// TwinCAT 3 PLC project cookie_module_shell
// ProgramVersion: 3.1.0.8
// libraries:
//   Tc2_Standard, * (Beckhoff Automation GmbH)
//   Tc2_System, * (Beckhoff Automation GmbH)
//   Tc3_Interfaces, * (Beckhoff Automation GmbH)
//   Tc3_Module, * (Beckhoff Automation GmbH)
//   Tc2_MC2,3.3.8.0,Beckhoff Automation GmbH
//   Tc2_TcpIp,3.3.2.0,Beckhoff Automation GmbH
//   Tc2_Utilities,3.3.7.0,Beckhoff Automation GmbH
// project tree:
//   DUTs/industrialPhysics/ MNG_APPLICATION_INPUTS_32BIT.TcDUT, MNG_APPLICATION_OUTPUTS_32BIT.TcDUT, MNG_DataArray.TcDUT (not stored), MNG_DatagramHeader.TcDUT (not stored), MNG_DatagramType.TcDUT (not stored), MNG_POSE6.TcDUT (not stored), MNG_RawDatagram.TcDUT (not stored), MNG_TRAFO.TcDUT (not stored), VEC3.TcDUT (not stored)
//   DUTs/InternalDataTypes/ eMainState.TcDUT, eSubState.TcDUT (not stored)
//   DUTs/OPC Interface/Server DUTs/ DUT_MODE.TcDUT, DUT_PARAMETER_INPUT.TcDUT, DUT_PARAMETER_OUTPUT.TcDUT, DUT_SERVER_MODULE_INTERFACE.TcDUT, DUT_SERVER_MODULE_INTERFACE_INPUT.TcDUT, DUT_SERVER_MODULE_INTERFACE_OUTPUT.TcDUT, DUT_SERVER_PARAMETERINPUTARRAY.TcDUT, DUT_SERVER_PARAMETEROUTPUTARRAY.TcDUT, DUT_SERVER_SKILLINPUTARRAY.TcDUT, DUT_SERVER_SKILLOUTPUTARRAY.TcDUT, DUT_SERVER_SKILL_INPUT.TcDUT, DUT_SERVER_SKILL_OUTPUT.TcDUT, DUT_SERVER_STATEVALUEARRAY.TcDUT, DUT_STATEVALUES.TcDUT
//   GVLs/ GVL.TcGVL, MI5.TcGVL, MNG_GLOBALS.TcGVL (not stored), OPCConstants.TcGVL
//   / PlcTask.TcTTO (not stored), SimuTask.TcTTO
//   POUs/ FB_EmergencyStop.TcPOU, FB_Error.TcPOU, FB_Init.TcPOU, FB_Output.TcPOU, FB_Ready.TcPOU, FB_Refill.TcPOU, FB_ResetSystem.TcPOU, FB_Separation.TcPOU, FB_Timer.TcPOU, FB_TurnDiskModulo.TcPOU, FB_TurnDiskToSensor.TcPOU, MAIN.TcPOU, FB_StorageLevel.TcPOU, FB_ResetAxis.TcPOU
//   POUs/industrialPhysics/ FB_LogFifo.TcPOU, MAIN_simu.TcPOU, MNG_SIMULATION.TcPOU, MNG_UPDATEIOS.TcPOU
// real-time tasks:
//   TASK PlcTask: cycle T#10ms, priority 20, ADS port 350
//   TASK SimuTask: cycle T#10ms, priority 21, ADS port 351
// motion (NC):
//   TASK NC-Task 1 SAF: cycle T#1ms, priority 4, ADS port 501
//   TASK NC-Task 1 SVB: cycle T#10ms, priority 8, ADS port 511
//   AXIS Axis 2 (id 2)
//     General: UnitName=Degree, UnitFlags=#x00000004
//     Dynamic: Acceleration=19710, Deceleration=19710, Jerk=59130
//     Velo: RefSearch=131.4, RefSync=131.4, SlowManual=657, FastManual=3942, Fast=13140, Maximum=13140
//     OtherSettings: AllowMotionCmdToSlave=true
//     encoder EncType=19
//       EncPara: ScaleFactorNumerator=360, ScaleFactorDenominator=1048576, MaxCount=#xffffffff
//         TimeComp: TimeCompMode=1
//     drive DrvType=16
//       DrvPara: MaxCount=#xffffffff
//         Analog: VeloReferenz=14454, VeloScale=32
//         TimeComp: TimeCompMode=1, TaskDelayCycles=1
//     controller CtrType=1
//       CtrPara: PriorControlFactor=1
//         PosDiffControl: Range=8, Time=0.3
//         PID: PosKp=25
//         Observer: BandWidth=20
// I/O:
//   DEVICE Device 1 (EtherCAT), AmsNetId 5.26.6.164.2.1
//     Term 1 (EK1200) [EK1200-5000 EtherCAT Power supply (2A E-Bus)]
//       Term 2 (EL1804) [EL1804 4Ch. Dig. Input 24V, 3ms]
//       Term 3 (EL2808) [EL2808 8Ch. Dig. Output 24V, 0.5A]
//       Term 4 (EL7211-0010) [EL7211-0010 1Ch. MDP742 Servo motor output stage with OCT (50V, 4.5A RMS)]
//       Term 5 (EK1110) [EK1110 EtherCAT extension]
//     Box 6 (ZAC50CN02 (Junction EtherCAT with PoE)) [ZAC50CN02 (Junction EtherCAT with PoE)]
//       Term 7 (Sub-Core 1 with two extern ports) [Sub-Core 1 with two extern ports]
//         Box 8 (OCPnnnP0150C) [OCPnnnP0150C Type 352]
//   DEVICE Device 3 (EtherCAT Automation Protocol) (disabled), AmsNetId 5.26.6.164.4.1
// variable links:
//   NC-Task 1 SAF/Axes/Axis 2 <-> Device 1 (EtherCAT)/Term 1 (EK1200)/Term 4 (EL7211-0010)
//     Enc/Inputs/In/nDataIn1 <-> FB Position/Position
//     Enc/Inputs/In/nDcInputTime <-> InfoData/DcInputShift
//     Drive/Inputs/In/nState1 <-> DRV Statusword/Statusword
//     Drive/Outputs/Out/nDataOut2 <-> DRV Target velocity/Target velocity
//     Drive/Inputs/In/nState2 <-> DRV Statusword/Statusword @bit 8
//     Drive/Inputs/In/nState4 @bit 1 <-> WcState/InputToggle
//     Enc/Inputs/In/nState4 @bit 1 <-> WcState/InputToggle
//     Drive/Inputs/In/nDcOutputTime <-> InfoData/DcOutputShift
//     Drive/Outputs/Out/nCtrl1 <-> DRV Controlword/Controlword
//     Enc/Inputs/In/nState4 <-> WcState/WcState
//     Drive/Outputs/Out/nCtrl2 <-> DRV Controlword/Controlword @bit 8
//     Drive/Inputs/In/nState4 <-> WcState/WcState
//   cookie_module_shell/cookie_module_shell Instance <-> Device 1 (EtherCAT)/Box 6 (ZAC50CN02 (Junction EtherCAT with PoE))
//     PlcTask Inputs/GVL.iDiskPosition <-> TxPDO/Read input 8 bit
//   cookie_module_shell/cookie_module_shell Instance <-> Device 1 (EtherCAT)/Box 6 (ZAC50CN02 (Junction EtherCAT with PoE))/Term 7 (Sub-Core 1 with two extern ports)/Box 8 (OCPnnnP0150C)
//     PlcTask Inputs/GVL.iStorageLevel <-> TxPDO/Measurement
//   cookie_module_shell/cookie_module_shell Instance <-> Device 1 (EtherCAT)/Term 1 (EK1200)/Term 2 (EL1804)
//     PlcTask Inputs/GVL.iCookieIntact <-> Channel 1/Input
//     PlcTask Inputs/GVL.iNoCookieInOutput <-> Channel 3/Input
//   cookie_module_shell/cookie_module_shell Instance <-> Device 1 (EtherCAT)/Term 1 (EK1200)/Term 3 (EL2808)
//     PlcTask Outputs/GVL.oTriggerCamera <-> Channel 1/Output
//   cookie_module_shell/cookie_module_shell Instance <-> NC-Task 1 SAF/Axes/Axis 2
//     PlcTask Inputs/GVL.axis.NcToPlc <-> Outputs/ToPlc
//     PlcTask Outputs/GVL.axis.PlcToNc <-> Inputs/FromPlc

CONFIGURATION cookie_module_shell
    RESOURCE PLC ON TwinCAT3
        TASK SimuTask(INTERVAL := T#10ms, PRIORITY := 21);
        PROGRAM MAIN_simu WITH SimuTask : MAIN_simu;
    END_RESOURCE
END_CONFIGURATION

// ---- DUTs/industrialPhysics/MNG_APPLICATION_INPUTS_32BIT.TcDUT

TYPE MNG_APPLICATION_INPUTS_32BIT :
STRUCT
    NumSignals                     : INT     := 5         ;
    HallSensor1_00_IR : BOOL    := 0; (* ysics/Keksmodul/Keksmodul - relevant/HallSensor1?IR *)
    HallSensor2_00_IR : BOOL    := 0; (* ysics/Keksmodul/Keksmodul - relevant/HallSensor2?IR *)
    init_sensor_cookie_module_00_IR : BOOL    := 0; (* l/Keksmodul - relevant/init_sensor_cookie_module?IR *)
    kein_cookie_mehr_00_IR : BOOL    := 0; (* /Keksmodul/Keksmodul - relevant/kein_cookie_mehr?IR *)
    cookiebox_sensor_00_IR : BOOL    := 0; (* Physics://physics/Keksmodul/cookiebox_sensor?IR *)
END_STRUCT
END_TYPE

// ---- DUTs/InternalDataTypes/eMainState.TcDUT
TYPE eMainState :
(
	init		:= 0,
	ready		:= 10,
	output		:= 20,
	separation	:= 30,
	refill		:= 40,
	emergencyStop	:= 50,
	error			:= 60,
	resetSystem		:= 70
);
END_TYPE

// ---- DUTs/industrialPhysics/MNG_APPLICATION_OUTPUTS_32BIT.TcDUT

TYPE MNG_APPLICATION_OUTPUTS_32BIT :
STRUCT
    NumSignals                     : INT     := 4         ;
    Disc_00_ACT_POS : REAL    := 0.0; (* ysics/Keksmodul/Keksmodul - relevant/Disc?KinActual *)
    A2014_09_12_Left_Predeterminado_00_ACT_POS : REAL    := 0.0; (* nt/Scissor/2014_09_12_Left_Predeterminado?KinActual *)
    A2014_09_12_Right_Predeterminado_00_ACT_POS : REAL    := 0.0; (* t/Scissor/2014_09_12_Right_Predeterminado?KinActual *)
    Keksquelle_00_TRIG02 : BOOL    := 0; (* Physics://physics/Keksmodul/Keksquelle?Trigger *)
END_STRUCT
END_TYPE

// ---- DUTs/OPC Interface/Server DUTs/DUT_MODE.TcDUT
/// MODE to run (inside of MODULE_INTERFACE_INPUT)
TYPE DUT_MODE :
(
	///Initialitzation number mode
	Init := 0,
	///Automatic number mode
	Auto := 1,
	///Manual number mode
	Manual := 2,
	Reset := 3
);
END_TYPE

// ---- DUTs/OPC Interface/Server DUTs/DUT_PARAMETER_INPUT.TcDUT
TYPE DUT_PARAMETER_INPUT :
STRUCT
	///Value of the parameter 
	Value: LREAL;
	///Possibility to a string value depending on the parameter
	StringValue: STRING(80);
END_STRUCT
END_TYPE

// ---- DUTs/OPC Interface/Server DUTs/DUT_PARAMETER_OUTPUT.TcDUT
TYPE DUT_PARAMETER_OUTPUT :
STRUCT
	///Free to use = TRUE, busy to use =FALSE
	Dummy: BOOL := TRUE;
	///ID of the parameter
	ID: UINT;
	///Name of the parameter
	Name: STRING(80);
	///Unit of the parameter
	Unit: STRING(80);
	///Optional parameter
	Required: BOOL;
	///Default parameter to work
	Default: LREAL;
	///Minimum value of the parameter
	MinValue: LREAL;
	///Maximum value of the parameter
	MaxValue: LREAL;
END_STRUCT
END_TYPE

// ---- DUTs/OPC Interface/Server DUTs/DUT_SERVER_MODULE_INTERFACE.TcDUT
/// MODULE INTERFACE INPUT AND OUTPUT 
TYPE DUT_SERVER_MODULE_INTERFACE :
STRUCT
	///Information that the module reads
	Input: DUT_SERVER_MODULE_INTERFACE_INPUT;
	///Information that the module write
	Output: DUT_SERVER_MODULE_INTERFACE_OUTPUT;
END_STRUCT
END_TYPE

// ---- DUTs/OPC Interface/Server DUTs/DUT_SERVER_MODULE_INTERFACE_INPUT.TcDUT
TYPE DUT_SERVER_MODULE_INTERFACE_INPUT :
STRUCT
	///Mode to run (init,auto,manual,..)
	Mode: INT;
	///check if the modules is alive
	ConnectionTestInput: BOOL;
	///Modules get their position
	PositionInput : LREAL;
	///Update data= TRUE, No updatedata=FALSE
	Watchbit: BOOL;
	///Emergency stop
	EmergencyStop: BOOL;
	///Range of INPUT skills
	SkillInput: DUT_SERVER_SKILLINPUTARRAY;
END_STRUCT
END_TYPE

// ---- DUTs/OPC Interface/Server DUTs/DUT_SERVER_MODULE_INTERFACE_OUTPUT.TcDUT
TYPE DUT_SERVER_MODULE_INTERFACE_OUTPUT :
STRUCT
	///Free to use = TRUE, busy to use =FALSE
	Dummy: BOOL := TRUE;
	///Individual name of the module
	Name: STRING(80);
	///Identification number of module
	ID: UINT;
	///IP address
	IP: STRING(80);
	///Show if the module is in Standby or not
	Idle: BOOL;
	///Show if the module is connected
	Connected: BOOL;
	///Feedback with conection test input
	ConnectionTestOutput: BOOL;
	///Show if the system has error when=TRUE
	Error: BOOL;
	///Identification number of the error
	ErrorID: UINT;
	///Description of the error
	ErrorDescription: STRING(80);
	///Description of the current task
	CurrentTaskDescription: STRING(80);
	///Position of the output
	PositionOutput: LREAL;
	/// Bool value of the Sensor
	PositionSensor: BOOL;
	///Range of OUTPUT skills
	SkillOutput: DUT_SERVER_SKILLOUTPUTARRAY;
	///Range of state values
	StateValue: DUT_SERVER_STATEVALUEARRAY;
END_STRUCT
END_TYPE

// ---- DUTs/OPC Interface/Server DUTs/DUT_SERVER_PARAMETERINPUTARRAY.TcDUT
TYPE DUT_SERVER_PARAMETERINPUTARRAY :
STRUCT
	ParameterInput0: DUT_PARAMETER_INPUT;
	ParameterInput1: DUT_PARAMETER_INPUT;
	ParameterInput2: DUT_PARAMETER_INPUT;
	ParameterInput3: DUT_PARAMETER_INPUT;
	ParameterInput4: DUT_PARAMETER_INPUT;
	ParameterInput5: DUT_PARAMETER_INPUT;
END_STRUCT
END_TYPE

// ---- DUTs/OPC Interface/Server DUTs/DUT_SERVER_PARAMETEROUTPUTARRAY.TcDUT
TYPE DUT_SERVER_PARAMETEROUTPUTARRAY :
STRUCT
	ParameterOutput0: DUT_PARAMETER_OUTPUT;
	ParameterOutput1: DUT_PARAMETER_OUTPUT;
	ParameterOutput2: DUT_PARAMETER_OUTPUT;
	ParameterOutput3: DUT_PARAMETER_OUTPUT;
	ParameterOutput4: DUT_PARAMETER_OUTPUT;
	ParameterOutput5: DUT_PARAMETER_OUTPUT;
END_STRUCT
END_TYPE

// ---- DUTs/OPC Interface/Server DUTs/DUT_SERVER_SKILLINPUTARRAY.TcDUT
TYPE DUT_SERVER_SKILLINPUTARRAY :
STRUCT
	SkillInput0: DUT_SERVER_SKILL_INPUT;
	SkillInput1: DUT_SERVER_SKILL_INPUT;
	SkillInput2: DUT_SERVER_SKILL_INPUT;
	SkillInput3: DUT_SERVER_SKILL_INPUT;
	SkillInput4: DUT_SERVER_SKILL_INPUT;
	SkillInput5: DUT_SERVER_SKILL_INPUT;
	SkillInput6: DUT_SERVER_SKILL_INPUT;
	SkillInput7: DUT_SERVER_SKILL_INPUT;
	SkillInput8: DUT_SERVER_SKILL_INPUT;
	SkillInput9: DUT_SERVER_SKILL_INPUT;
	SkillInput10: DUT_SERVER_SKILL_INPUT;
	SkillInput11: DUT_SERVER_SKILL_INPUT;
	SkillInput12: DUT_SERVER_SKILL_INPUT;
	SkillInput13: DUT_SERVER_SKILL_INPUT;
	SkillInput14: DUT_SERVER_SKILL_INPUT;
	SkillInput15: DUT_SERVER_SKILL_INPUT;
END_STRUCT
END_TYPE

// ---- DUTs/OPC Interface/Server DUTs/DUT_SERVER_SKILLOUTPUTARRAY.TcDUT
TYPE DUT_SERVER_SKILLOUTPUTARRAY :
STRUCT
	SkillOutput0: DUT_SERVER_SKILL_OUTPUT;
	SkillOutput1: DUT_SERVER_SKILL_OUTPUT;
	SkillOutput2: DUT_SERVER_SKILL_OUTPUT;
	SkillOutput3: DUT_SERVER_SKILL_OUTPUT;
	SkillOutput4: DUT_SERVER_SKILL_OUTPUT;
	SkillOutput5: DUT_SERVER_SKILL_OUTPUT;
	SkillOutput6: DUT_SERVER_SKILL_OUTPUT;
	SkillOutput7: DUT_SERVER_SKILL_OUTPUT;
	SkillOutput8: DUT_SERVER_SKILL_OUTPUT;
	SkillOutput9: DUT_SERVER_SKILL_OUTPUT;
	SkillOutput10: DUT_SERVER_SKILL_OUTPUT;
	SkillOutput11: DUT_SERVER_SKILL_OUTPUT;
	SkillOutput12: DUT_SERVER_SKILL_OUTPUT;
	SkillOutput13: DUT_SERVER_SKILL_OUTPUT;
	SkillOutput14: DUT_SERVER_SKILL_OUTPUT;
	SkillOutput15: DUT_SERVER_SKILL_OUTPUT;
END_STRUCT
END_TYPE

// ---- DUTs/OPC Interface/Server DUTs/DUT_SERVER_SKILL_INPUT.TcDUT
TYPE DUT_SERVER_SKILL_INPUT :
STRUCT
	///Range of parameters
	ParameterInput: DUT_SERVER_PARAMETERINPUTARRAY;
	///Start process
	Execute: BOOL;
END_STRUCT
END_TYPE

// ---- DUTs/OPC Interface/Server DUTs/DUT_SERVER_SKILL_OUTPUT.TcDUT
TYPE DUT_SERVER_SKILL_OUTPUT :
STRUCT
	///Free to use = TRUE, busy to use =FALSE
	Dummy: BOOL := TRUE;
	///Identification number of skill
	ID: UINT;
	///indentfication name of skill
	Name: STRING(80);
	///Skill activated
	Activated: BOOL;
	///Ready to do skill
	Ready: BOOL;
	///Skill in process
	Busy: BOOL;
	///Skill finish
	Done: BOOL;
	///Error in system
	Error: BOOL;
	///Range of parameters
	ParameterOutput: DUT_SERVER_PARAMETEROUTPUTARRAY;
END_STRUCT
END_TYPE

// ---- DUTs/OPC Interface/Server DUTs/DUT_SERVER_STATEVALUEARRAY.TcDUT
TYPE DUT_SERVER_STATEVALUEARRAY :
STRUCT
	StateValue0: DUT_STATEVALUES;
	StateValue1: DUT_STATEVALUES;
	StateValue2: DUT_STATEVALUES;
	StateValue3: DUT_STATEVALUES;
	StateValue4: DUT_STATEVALUES;
	StateValue5: DUT_STATEVALUES;
	StateValue6: DUT_STATEVALUES;
	StateValue7: DUT_STATEVALUES;
	StateValue8: DUT_STATEVALUES;
	StateValue9: DUT_STATEVALUES;
	StateValue10: DUT_STATEVALUES;
END_STRUCT
END_TYPE

// ---- DUTs/OPC Interface/Server DUTs/DUT_STATEVALUES.TcDUT
TYPE DUT_STATEVALUES :
STRUCT
	///Free to use = TRUE, busy to use =FALSE
	Dummy: BOOL := TRUE;
	///Value of the State
	Value: LREAL;
	///Name of the state
	Name: STRING(80);
	///Description of the state
	Description: STRING(80);
	///Unit of the state ()
	Unit: STRING(80);
END_STRUCT
END_TYPE

// ---- GVLs/GVL.TcGVL
VAR_GLOBAL
	pi : REAL := 3.14159;
																
	//<<Input Variables>>//
	//iExecute				AT%I*	: BOOL; 			// is there a order to separate cookies? --> from database
	//iClearence			AT%I*	: BOOL;				// did the user clear the refilling/maintenance process --> from HMI
														//@TODO: change to Mode change? mode: init, auto, manual
	//iEmergencyStop		AT%I*	: BOOL;				// stop all running tasks and transform the machine in a safe state
	
	iDiskPosition 		AT%I*	: INT; 				// is the gap of the disk at the storage? --> 2 the ramp? --> 1 --> from hall sensor
	iNoCookieInOutput	AT%I*	: BOOL;				// is the cookie in the ouput (on the clamp)? --> from light barrier sensor
	iStorageLevel 		AT%I*	: DINT;			// number of remaining cookies in the storage --> from distance sensor
	iCookieIntact		AT%I*	: BOOL;				// camera detection if cookie intact or broken
	

	//<<Output Variables>>//
	oTriggerCamera		AT%Q*	: BOOL	:= FALSE;	//Variable to init the flashing mode of the cam		
	
	//<<Internal Variables>>//
	mainState 					: eMainState		:= eMainState.init;
	refillSubState				: eSubState			:= eSubState.step0;
	separationSubState			: eSubState			:= eSubstate.step0;
	initSubState				: eSubState			:= eSubstate.step0;
	outputSubState				: eSubState			:= eSubstate.step0;
	emergencySubState			: eSubState			:= eSubstate.step0;
	errorSubState				: eSubState			:= eSubstate.step0;
	resetSubState				: eSubState			:= eSubstate.step0;

	axis	 					: AXIS_REF;
	empty						: BOOL;				// is cookie storage empty
	fastVel						: INT	:= 40;		//@TODO: Use something to change velocity in ParameterInput
	slowVel						: INT	:= 15;		//@TODO: Use something to change velocity in ParameterInput
	
	modulePositionInitialized	: BOOL := FALSE;	// is the module position initialized
	firstRun					: BOOL := TRUE;		// is this the first init? then wait for axis to get ready
	
	
	//<<For Simulation>>//
	offset						: LREAL;
	infinitsimu					: BOOL;
	infinitsimu2				: BOOL;
	init_sensor 				: BOOL;      //AT	%I*, muss vor :BOOL ,Änderung km
	SensorPosition				: LREAL;				
	
END_VAR

// ---- GVLs/MI5.TcGVL
VAR_GLOBAL
	//<<OPC-UA Module Interface>>//
	{attribute 'OPC.UA.DA' := '1'}
	Module2101 : DUT_SERVER_MODULE_INTERFACE;
	{attribute 'OPC.UA.DA' := '1'}
	reset : BOOL := FALSE;
	{attribute 'OPC.UA.DA' := '1'}
	cameraFix : BOOL := FALSE;
END_VAR

// ---- GVLs/OPCConstants.TcGVL
VAR_GLOBAL CONSTANT
	///Maximum number of skillparameters
	ParameterCnt: INT := 5;
	///Maximum number of skills per Module
	SkillCnt: INT := 15;
	///Maximum number of Statevalues of one Module
	StateCnt: INT := 10;
	///Maximum number of modules
	ModuleCnt: INT := 10;
	///Maximum number of Tasks in Production List
	TaskCnt: INT := 30;
	///Maximum number  of offered recipes
	OfferCnt: INT := 5;
	///Maximum number of Orders in Queue
	OrderCnt: INT := 5;
	///Number of user set parameters per recipe
	UserParameterCnt: INT := 5;
	///Number of skills per task
	TaskSkillCnt: INT := 50;
END_VAR

// ---- POUs/industrialPhysics/MAIN_simu.TcPOU

PROGRAM MAIN_simu
VAR
    simIO : MNG_Simulation;
END_VAR

// Update IOs with simulation
simIO(bEnable := TRUE);

// Application code follows here:

END_PROGRAM

// ---- POUs/industrialPhysics/MNG_SIMULATION.TcPOU
FUNCTION_BLOCK MNG_Simulation
VAR_INPUT
    bEnable    : BOOL                          := FALSE;
    outputs AT %I*   : MNG_Application_Outputs_32Bit         ;
END_VAR
VAR_OUTPUT
    inputs AT %Q*  : MNG_Application_Inputs_32Bit          ;
END_VAR
VAR
    ioUpdater  : MNG_UpdateIOs                 := (sRemoteHost := '192.168.42.31', nRemotePort := 5110);
    fbCloseAll : FB_SocketCloseAll;
    bCloseAll  : BOOL := TRUE;
	trig		: BOOL;
END_VAR

(* @END_DECLARATION := '0'                                                    *)
IF bCloseAll THEN (*On PLC reset or program download close all old (opened) connections *)
    bCloseAll := FALSE;
    fbCloseAll( bExecute:= TRUE );
ELSE
    fbCloseAll( bExecute:= FALSE );
END_IF

IF NOT fbCloseAll.bBusy THEN

    (* ------------------------------------- trigger data exchange ----------------------------------------------------------------------------*)
    ioUpdater(Outputs := outputs, Inputs := inputs, bEnable := bEnable);

END_IF

// Application code follows here:

{*IF GVL.infinitsimu THEN
	outputs.Disc_00_ACT_POS := (REAL_TO_INT(GVL.SensorPosition -180 + GVL.axis.NcToPlc.ModuloActPos))MOD 360;
ELSE
	IF GVL.infinitsimu2 THEN
		outputs.Disc_00_ACT_POS := (REAL_TO_INT(GVL.SensorPosition + GVL.axis.NcToPlc.ModuloActPos))MOD 360;
	ELSE
		outputs.Disc_00_ACT_POS := GVL.axis.NcToPlc.ModuloActPos;
	END_IF	
END_IF*}

outputs.Disc_00_ACT_POS := GVL.axis.NcToPlc.ModuloSetPos;

//storageLevel.full := inputs.kein_cookie_mehr_00_IR;

outputs.A2014_09_12_Right_Predeterminado_00_ACT_POS := ABS(SIN(((GVL.axis.NcToPlc.ActPos*pi)/180)))*(-7);
outputs.A2014_09_12_Left_Predeterminado_00_ACT_POS := ABS(SIN(((GVL.axis.NcToPlc.ActPos*pi)/180)))*(7);

//GVL.iNoCookieInOutput := inputs.cookiebox_sensor_00_IR;
//GVL.iDiskAtStorage := inputs.HallSensor1_00_IR;
//GVL.iDiskAtRamp := inputs.HallSensor2_00_IR;

GVL.init_sensor := inputs.cookiebox_sensor_00_IR;

IF GVL.mainState = eMainState.ready THEN
	trig := TRUE;
ELSE 
	trig := FALSE;
END_IF

//trigger(CLK:= trig, Q=> newCookie);
IF trig THEN
	outputs.Keksquelle_00_TRIG02 := TRUE;
ELSE 
	outputs.Keksquelle_00_TRIG02 := FALSE;
END_IF 


//outputs.Keksquelle_00_ReleaseTime := 60;
//outputs.Keksquelle_00_AlwaysOn := TRUE;

END_FUNCTION_BLOCK

// ---- POUs/industrialPhysics/MNG_UPDATEIOS.TcPOU
FUNCTION_BLOCK MNG_UpdateIOs
(* This function block implements simple TCP/IP client protocol.              *)
(* The max. size of binary tx/rx data has to be <= PLCPRJ_BUFFER_SIZE         *)
VAR_IN_OUT
    Outputs : MNG_Application_Outputs_32Bit;    (* Tx user data *)
    Inputs      : MNG_Application_Inputs_32Bit                        ; (* Rx user data *)
END_VAR

VAR_INPUT
    bDbg        : BOOL                         := FALSE               ; (* TRUE => Enable debug output, FALSE => Disable debug output *)
    sRemoteHost : STRING(15)                   := '127.0.0.1'         ; (* IP address of remote server *)	
    nRemotePort : UDINT                        := 5000                ; (* Remote server port *)
    bEnable     : BOOL                         := FALSE               ; (* TRUE => Enable/connect, FALSE => Disable/disconnect *)
    tReconnect  : TIME                         := T#5s                ;
END_VAR

VAR_OUTPUT
    errors      : FB_LogFifo                                          ; (* Error message fifo *)
    eState      : E_SocketConnectionState      := eSOCKET_DISCONNECTED; (* TCP/IP connection state *)
END_VAR

VAR
    counter          : DWORD                        := 0                   ;
    fbConnect        : FB_ClientServerConnection    := (tReconnect := T#5s); (* Create/release TCP/IP connection *)
    fbSend           : FB_SocketSend                                       ; (* Send TCP/IP data *)
    fbReceive        : FB_SocketReceive                                    ; (* Receive TCP/IP data *)
    state            : BYTE                                                ; (* Global state *)
    tx_state         : BYTE                                                ; (* Tx state *)
    rx_state         : BYTE                                                ; (* Rx state *)

    toServer         : MNG_RawDatagram                                     ;
    fromServer       : MNG_RawDatagram                                     ;
    cbReceived       : UDINT                                               ; (* Count of received data bytes *)
    cbRx             : UDINT                                               ; (* Rx frame byte size *)

    bDisconnect      : BOOL                                                ; (* Disconnect flag, if set the socket will be closed *)
    pollTimer        : TON                                                 ; (* Rx data poll timer *)
    bAbort           : BOOL                                                ; (* Flag to abort frame parsing loop *)
    sID              : STRING(20)                   := ''                  ;
    clock            : FB_LocalSystemTime           := ( bEnable := TRUE ) ; (* OS clock *)
    _byteCount       : DWORD                                               ;
    _i               : DWORD                                               ;
    _ptr             : POINTER TO BYTE                                     ;
    _internalInputs  : MNG_Application_Inputs_32Bit                        ;
    DWordBuffer      : DWORD                                               ; (* convert DWORD data *)
    DIntBuffer       : DINT                                                ; (* convert DINT data *)
END_VAR


(* refresh clock time                                                         *)
clock();

(* state chart                                                                *)
CASE state OF
    0:(* Init state *)
        (*rx.A_Reset(bDbg := bDbg)  ; (* Reset RX fifo (optional) *)
        tx.A_Reset    (bDbg := bDbg); (* Reset TX fifo (optional) *)*)
        errors.Clear(); (* Reset error fifo (optional) *)

        pollTimer( IN := FALSE, PT := PLCPRJ_RECEIVER_POLLING_CYCLE_TIME );
        bDisconnect := FALSE;(* Reset disconnect flag *)
        cbReceived  := 0;(* Reset number of received data bytes *)
        tx_state    := 0;(* Reset tx state machine *)
        rx_state    := 0;(* Reset rx state machine *)
        state       := 1;(* Go to the next step *)

    1:(* Create TCP/IP connection *)
        fbConnect(sSrvNetID := '',
                  nMode := CONNECT_MODE_ENABLEDBG,(* Enable debug output *)
                  sRemoteHost := sRemoteHost,
                  nRemotePort := nRemotePort,
                  tReconnect  := tReconnect,
                  bEnable     := bEnable,
                  eState      => eState);
        IF NOT fbConnect.bBusy THEN

            (* Create identification string used by debug messages *)
            sID          := CONCAT(CONCAT('[', DWORD_TO_HEXSTR(fbConnect.hSocket.handle, 4, FALSE) ), ']');
            errors.sMessage := CONCAT('CLI.Err', sID);

            IF NOT fbConnect.bError THEN
                IF eState = eSOCKET_CONNECTED THEN(* we are connected *)
                    state := 2;
                END_IF
            ELSE(* connect error: log error *)
                errors.Error(nErrId := fbConnect.nErrId);
            END_IF
        END_IF

    2:(* Data exchange state *)
        bDisconnect := NOT bEnable OR bDisconnect; (* user/internal disconnect requested? *)
        IF bDisconnect AND (tx_state = 0) AND (rx_state = 0) THEN
            state := 3;(* disconnect *)
        ELSE
            (*--------------------------- Send tx data -------------------------------------------*)
            CASE tx_state OF
                0:
                    IF NOT bDisconnect THEN

                        (* forcefully send data each cycle *)

                        (* create the raw datagram *)
                        _byteCount                   := 20;
                        toServer.Header.ByteCount    := HOST_TO_BE32(in := _byteCount);
                        toServer.Header.DatagramType := HOST_TO_BE32(in := MNG_Raw32BitImage);
                        toServer.Header.Counter      := Counter;

                        toServer.Payload[1] := HOST_TO_BE32(4); (* number of signals *)

                        (* FLOAT32 Disc_00_ACT_POS *)
                        MEMCPY(destAddr := ADR(DWordBuffer), srcAddr := ADR(Outputs.Disc_00_ACT_POS), n := 4);
                        toServer.Payload[2] := HOST_TO_BE32(DWordBuffer);

                        (* FLOAT32 A2014_09_12_Left_Predeterminado_00_ACT_POS *)
                        MEMCPY(destAddr := ADR(DWordBuffer), srcAddr := ADR(Outputs.A2014_09_12_Left_Predeterminado_00_ACT_POS), n := 4);
                        toServer.Payload[3] := HOST_TO_BE32(DWordBuffer);

                        (* FLOAT32 A2014_09_12_Right_Predeterminado_00_ACT_POS *)
                        MEMCPY(destAddr := ADR(DWordBuffer), srcAddr := ADR(Outputs.A2014_09_12_Right_Predeterminado_00_ACT_POS), n := 4);
                        toServer.Payload[4] := HOST_TO_BE32(DWordBuffer);

                        (* BOOL Keksquelle_00_TRIG02 *)
                        IF Outputs.Keksquelle_00_TRIG02 THEN
                            toServer.Payload[5] := 16#FFFFFFFF;   (*BOOL *)
                        ELSE
                            toServer.Payload[5] := 0;
                        END_IF;

                        toServer.Header.SentTime := HOST_TO_BE32(in := clock.systemTime.wMilliseconds + clock.systemTime.wMinute * 60000);

                        (* send frame *)
                        fbSend(bExecute  := FALSE);
                        fbSend(sSrvNetID := '',
                               hSocket   := fbConnect.hSocket,
                               cbLen     := SIZEOF(toServer.Header) + _byteCount,(* size of header + size of user data *)
                               pSrc      := ADR(toServer),(* pointer to the frame data *)
                               bExecute  := TRUE,
                               tTimeout  := T#5s);

                        tx_state := 1;
                    END_IF
                1:(* wait until send not busy *)
                    fbSend( bExecute := FALSE );
                    IF NOT fbSend.bBusy THEN
                        tx_state := 0;
                        IF NOT fbSend.bError THEN(* no error *)
                            ;
                        ELSE(* send error => log error and disconnect *)
                            errors.Error(nErrId := fbSend.nErrId );
                            bDisconnect := TRUE;(* set flag *)
                        END_IF
                    END_IF
            END_CASE

            (* ------------------------------------------- Get/fetch rx data ----------------------------------------------------------------- *)
            CASE rx_state OF
                0:
                    IF NOT bDisconnect THEN
                        pollTimer( IN := TRUE );
                        IF pollTimer.Q THEN
                            pollTimer( IN := FALSE );

                            fbReceive( bExecute := FALSE );
                            fbReceive( 	sSrvNetId	:= '',
                            hSocket		:= fbConnect.hSocket,
                            cbLen		:= SIZEOF(fromServer) - cbReceived,
                            pDest		:= ADR(fromServer) + cbReceived,
                            bExecute	:= TRUE,
                            tTimeout	:= T#5s );
                            rx_state := 1;
                        END_IF
                    END_IF
                1:(* wait until receive not busy *)
                    fbReceive( bExecute := FALSE );
                    IF NOT fbReceive.bBusy THEN
                        rx_state := 0;
                        IF NOT fbReceive.bError THEN
                            IF fbReceive.nRecBytes > 0 THEN (* some bytes received *)

                                pollTimer( PT := T#0s );(* increase polling speed *)
                                cbReceived := cbReceived + fbReceive.nRecBytes;

                                (* parse received bytes *)
                                REPEAT
                                    bAbort := TRUE;(* set flag *)
                                    IF cbReceived >= SIZEOF(fromServer.Header) THEN (* all header bytes received => check header data *)

                                        (* correct header data *)
                                        fromServer.Header.ByteCount    := BE32_TO_HOST(fromServer.Header.ByteCount);
                                        Counter                        := fromServer.Header.Counter;
                                        fromServer.Header.SentTime     := BE32_TO_HOST(fromServer.Header.SentTime);
                                        fromServer.Header.DatagramType := BE32_TO_HOST(fromServer.Header.DatagramType);

                                        IF (fromServer.Header.ByteCount <= SIZEOF( fromServer.Payload))(* check frame (user data) length *)
                                        THEN

                                            cbRx := SIZEOF(fromServer.Header) + fromServer.Header.ByteCount;(* calculate the (expected) length of the rx frame *)
                                            IF cbReceived >= cbRx  THEN (* all frame bytes received? *)

                                               (* currently only use the data on a 32 Bit raw image *)
                                                IF fromServer.Header.DatagramType = MNG_Raw32BitImage THEN

                                                    IF 20 = (fromServer.Header.ByteCount - 4) THEN

                                                        (* BOOL HallSensor1_00_IR *)
                                                        Inputs.HallSensor1_00_IR := fromServer.Payload[2]<>0;

                                                        (* BOOL HallSensor2_00_IR *)
                                                        Inputs.HallSensor2_00_IR := fromServer.Payload[3]<>0;

                                                        (* BOOL init_sensor_cookie_module_00_IR *)
                                                        Inputs.init_sensor_cookie_module_00_IR := fromServer.Payload[4]<>0;

                                                        (* BOOL kein_cookie_mehr_00_IR *)
                                                        Inputs.kein_cookie_mehr_00_IR := fromServer.Payload[5]<>0;

                                                        (* BOOL cookiebox_sensor_00_IR *)
                                                        Inputs.cookiebox_sensor_00_IR := fromServer.Payload[6]<>0;

                                                    ELSE(* receive error: invalid frame format/data *)
                                                        errors.Error(nErrId := PLCPRJ_ERROR_INVALID_IO_FORMAT_RECEIVED );
                                                    END_IF

                                                END_IF

                                                MEMMOVE( ADR( fromServer ), ADR( fromServer ) + cbRx,  cbReceived - cbRx );(* shift the remaining rx bytes *)
                                                cbReceived := cbReceived - cbRx;(* recalculate the size of the remaining rx bytes *)

                                                bAbort := FALSE;(* reset flag, try to parse next frame *)

                                                (* ELSE repeat reading *)
                                            END_IF

                                        ELSE(* receive error: invalid frame format/data *)
                                            errors.Error(nErrId := PLCPRJ_ERROR_INVALID_FRAME_FORMAT );
                                            bDisconnect := TRUE;(* set flag *)
                                        END_IF
                                        (* ELSE repeat reading *)
                                    END_IF (* IF cbReceived >= SIZEOF(rxFrame.head) THEN *)

                                UNTIL bAbort
                                END_REPEAT

                            ELSE(* fbReceive.nRecBytes = 0, repeat reading *)
                                pollTimer( PT := PLCPRJ_RECEIVER_POLLING_CYCLE_TIME );(* slow down the polling cycle *)
                            END_IF(* IF fbReceive.nRecBytes > 0 THEN *)
                        ELSE(* receive error => log error and disconnect *)
                            errors.Error(nErrId := fbReceive.nErrId );
                            bDisconnect := TRUE;(* set flag *)
                        END_IF

                    END_IF(*IF NOT fbReceive.bBusy THEN*)

            END_CASE

        END_IF

    3:(* disconnect *)
        fbConnect( bEnable:= FALSE, eState=>eState );
        IF eState = eSOCKET_DISCONNECTED THEN
            state := 0;
        END_IF

END_CASE

END_FUNCTION_BLOCK

// ---- POUs/industrialPhysics/FB_LogFifo.TcPOU
(* Log/debug/error message fifo *)
FUNCTION_BLOCK FB_LogFifo
VAR_INPUT
	bLog		: BOOL 		:= FALSE;(* TRUE => Enable log message output, FALSE => Disable *)
	sPrefix		: STRING 	:= 'Unknown::';(* Log message description string (allows the identification of log message source) *)
	
	sMessage	: STRING 	:= '';(* String message to add (write) to the fifo *)
	nErrID		: UDINT 	:= 0;(* Error code to add (write) to the fifo *)
	hSocket		: T_HSOCKET;(* Socket connection handle *)
END_VAR
VAR_OUTPUT
	bOk			: BOOL;(* TRUE = New entry added or removed succesfully, FALSE = Fifo overflow or fifo empty *)
	sGet		: T_MaxString := '';(* String entry removed (read) from fifo *)
	nCount		: UDINT := 0;(* Number of fifo entries *)
END_VAR
VAR
	fbBuffer 	: FB_StringRingBuffer;(* Basic (lower level) string buffer control function block *)
	buffer		: ARRAY[0..PLCPRJ_BUFFER_SIZE] OF BYTE;(* Internal buffer memory *)
	sSource		: T_MaxString;	
	sPut		: T_MaxString;
END_VAR

;

ACTION Error:
(* Adds new fifo entry *)
IF nErrID = 0 THEN
	sSource := '::Error: 0x';
ELSIF ( nErrID AND 16#80000000) = 16#80000000 THEN
	IF nErrID = 16#80072746 THEN
		sSource := '::Win32 error (the connection is reset by remote side): 0x';
	ELSE
		sSource := '::Win32 error: 0x';
	END_IF
ELSIF (nErrID AND 16#00008100) = 16#00008100 THEN
	CASE nErrID OF
		PLCPRJ_ERROR_RECEIVE_TIMEOUT:
			sSource := '::PLC sample project receive timeout error: 0x';
		PLCPRJ_ERROR_SENDFIFO_OVERFLOW:
			sSource := '::PLC sample project send fifo overflow error: 0x';
		PLCPRJ_ERROR_RECFIFO_OVERFLOW:
			sSource := '::PLC sample project receive fifo overflow error: 0x';
		PLCPRJ_ERROR_INVALID_FRAME_FORMAT:
			sSource := '::PLC sample project invalid frame format error: 0x';
	ELSE
		sSource := '::Other PLC sample project error: 0x';
	END_CASE
ELSIF (nErrID AND 16#00008000) = 16#00008000 THEN
	sSource := '::Internal TCP/IP Connection Server error: 0x';
ELSE
	sSource := '::TwinCAT System error: 0x';
END_IF

sPut := CONCAT( CONCAT( CONCAT( sPrefix, sMessage ), sSource ), DWORD_TO_HEXSTR( nErrID AND 16#FFFF, 0, FALSE ) ); 

fbBuffer.A_AddTail( pBuffer:= ADR(buffer), cbBuffer:= SIZEOF(buffer),
					putValue:= sPut, bOk=>bOk, nCount=>nCount );
IF bOk THEN
	IF bLog THEN(* Log error message *)
		ADSLOGSTR( ADSLOG_MSGTYPE_ERROR OR ADSLOG_MSGTYPE_LOG, '%s', sPut );	
	END_IF
END_IF
END_ACTION

ACTION Message:
(* Adds new fifo entry *)
sPut := CONCAT( CONCAT( sPrefix, sMessage ), CONCAT( '::', HSOCKET_TO_STRING(hSocket) ) );
fbBuffer.A_AddTail( pBuffer:= ADR(buffer), cbBuffer:= SIZEOF(buffer),
					putValue:= sPut, bOk=>bOk, nCount=>nCount );
IF bOk THEN
	IF bLog THEN(* Log information message *)
		ADSLOGSTR( ADSLOG_MSGTYPE_HINT OR ADSLOG_MSGTYPE_LOG, '%s', sPut );	
	END_IF
END_IF
END_ACTION

ACTION Remove:
(* Removes oldest fifo entry *)
IF nCount = 0 THEN
	sGet := '';
	bOk := FALSE;
	RETURN;
END_IF

fbBuffer.A_RemoveHead( pBuffer:= ADR(buffer), cbBuffer:= SIZEOF(buffer),
						getValue=>sGet, bOk=>bOk, nCount=>nCount );
END_ACTION

ACTION Clear:
(* Clears all fifo entries *)
fbBuffer.A_Reset( 	pBuffer := ADR( buffer ), cbBuffer := SIZEOF( buffer ), 
					bOk=>bOk, nCount=>nCount, getValue=>sGet );
END_ACTION

END_FUNCTION_BLOCK

// ---- POUs/FB_EmergencyStop.TcPOU
FUNCTION_BLOCK FB_EmergencyStop
VAR_INPUT
END_VAR
VAR_OUTPUT
END_VAR
VAR
END_VAR

CASE emergencySubState OF

	step0:	//setting of OPCUA variables
			Module2101.Output.SkillOutput.SkillOutput0.Busy := FALSE;
			Module2101.Output.SkillOutput.SkillOutput0.Done := FALSE;
			Module2101.Output.SkillOutput.SkillOutput0.Dummy := FALSE;
			Module2101.Output.SkillOutput.SkillOutput0.Error := TRUE;
			Module2101.Output.SkillOutput.SkillOutput0.Ready := FALSE;
			//go into the right error state
			Module2101.Output.ErrorID := 2;
			Module2101.Output.CurrentTaskDescription := 'Emergency stop';
			Module2101.Output.Error := TRUE;
			Module2101.Output.ErrorDescription := 'Emergency stop';
			
			//wait for process tool to set the module in manual mode
			IF(Module2101.Input.Mode = DUT_MODE.Manual) THEN
				emergencySubState := step1;
			END_IF
			
	step1:	//wait for process tool to set the module in init mode
			IF(Module2101.Input.Mode = DUT_MODE.Auto) THEN
				//reset error 
				Module2101.Output.Error := FALSE;
				Module2101.Output.ErrorDescription := '';
				Module2101.Output.ErrorID := 0;
				
				//change to init state
				initSubState := step0;
				mainState := eMainState.init;
				emergencySubState := step0;
			END_IF
			
			
	step2:	
			
	step3:	

END_CASE

END_FUNCTION_BLOCK

// ---- POUs/FB_Error.TcPOU
FUNCTION_BLOCK FB_Error
VAR_INPUT
END_VAR
VAR_OUTPUT
END_VAR
VAR
	resetAxis			: FB_ResetAxis;
END_VAR

//@TODO: implement all possible errors

CASE errorSubState OF

	step0:	Module2101.Output.SkillOutput.SkillOutput0.Busy := FALSE;
			Module2101.Output.SkillOutput.SkillOutput0.Done := FALSE;
			Module2101.Output.SkillOutput.SkillOutput0.Dummy := FALSE;
			Module2101.Output.SkillOutput.SkillOutput0.Error := TRUE;
			Module2101.Output.SkillOutput.SkillOutput0.Ready := FALSE;
			
			// Error: axis got stuck
			IF (axis.Status.ErrorID = 17744) THEN
				Module2101.Output.ErrorDescription := 'Axis got stuck. Please clear module.';
				Module2101.Output.ErrorID := 101;
				errorSubState := step1;
			END_IF
			
			IF (Module2101.Output.ErrorID = 0) THEN
				Module2101.Output.ErrorDescription := 'Unknown Error.';
				Module2101.Output.ErrorID := 199;
				errorSubState := step1;
			END_IF
			
			//change in the right error state
			Module2101.Output.CurrentTaskDescription := 'Error';
			Module2101.Output.Error := TRUE;
			
	step1:	//wait for process tool to set the module in manual mode
			IF(Module2101.Input.Mode = DUT_MODE.Manual) THEN
				resetAxis(execute:= FALSE);
				errorSubState := step2;
			END_IF
			
	step2:	IF NOT resetAxis.done THEN
				// axreset
				resetAxis (execute := TRUE);
			ELSE			
				errorSubState := step3;
			END_IF
			
	step3:	//wait for process tool to set the module in init mode
			IF(Module2101.Input.Mode = DUT_MODE.Auto) THEN
				
				//reset error 
				Module2101.Output.Error := FALSE;
				Module2101.Output.ErrorDescription := '';
				Module2101.Output.ErrorID := 0;
				
				//change to init state
				initSubState := step0;
				errorSubState := step0;
				mainState := eMainState.init;				
			END_IF
END_CASE

END_FUNCTION_BLOCK

// ---- POUs/FB_ResetAxis.TcPOU
FUNCTION_BLOCK FB_ResetAxis
VAR_INPUT
	execute: BOOL;
END_VAR
VAR_OUTPUT
	done : BOOL;
	busy : BOOL;
	error: BOOL;
END_VAR
VAR
	state			: INT := 0;
	fbreset			: Tc2_MC2.MC_Reset;
END_VAR

IF execute THEN
	CASE state OF
	
	0: 
		done := FALSE;
		fbreset(axis := axis, Execute := FALSE);
		state := 1;
		
	1:
		fbreset(
				Axis:= axis, 
				Execute:= TRUE, 
				Done=> , 
				Busy=> , 
				Error=> error, 
				ErrorID=> );
		IF fbreset.Done THEN
			state := 2;
		END_IF
		
	2:	
		execute := FALSE;
		done  := TRUE;
		state := 0;

	END_CASE
ELSE
	done := FALSE;
	state := 0;
END_IF

END_FUNCTION_BLOCK

// ---- POUs/FB_Init.TcPOU
FUNCTION_BLOCK FB_Init
VAR_INPUT
END_VAR
VAR_OUTPUT	
END_VAR
VAR
	turnDiskSensor	: FB_TurnDiskToSensor;		//turns disk to next sensor anti-clockwise
	turnDiskMod		: FB_TurnDiskModulo;		//turns disk back due to lag while stopping
	setPosition		: Tc2_MC2.MC_SetPosition;	//for initializing the motor position to a certain value
	resetAxis		: FB_ResetAxis;
	timer			: FB_Timer;
END_VAR

CASE initSubState OF 
	
	step0:	// wait for everything to boot in first run
			IF (firstRun) THEN
				timer(iTime:=T#5S, execute := TRUE);
				IF(timer.done) THEN
					firstRun := FALSE;
				END_IF
			ELSE
				initSubState := step1;
			END_IF

	step1:	turnDiskSensor(execute:= FALSE);
			resetAxis(execute:= FALSE);
			
			//reset all substates
			refillSubState := step0;
			separationSubState := step0;
			outputSubState := step0;
			emergencySubState := step0;
			errorSubState := step0;
			
			//>>>OPCUA Init<<<
	
			//>Modules<:
			Module2101.Output.ID := 2101;
			Module2101.Output.Name := 'Cookie Seperator';
			Module2101.Output.IP := '192.168.175.213';
			Module2101.Output.CurrentTaskDescription := 'Init process started: OPC UA';
			Module2101.Output.Dummy := FALSE;
			Module2101.Output.Idle  := FALSE;
			Module2101.Output.Error := FALSE;
			Module2101.Output.ErrorDescription := '';
			Module2101.Output.ErrorID := 0;
					
			//>Skill<: [0]=separate cookie
			Module2101.Output.SkillOutput.SkillOutput0.ID := 1010;
			Module2101.Output.SkillOutput.SkillOutput0.Activated := TRUE;
			Module2101.Output.SkillOutput.SkillOutput0.Busy := TRUE;
			Module2101.Output.SkillOutput.SkillOutput0.Done := FALSE;
			Module2101.Output.SkillOutput.SkillOutput0.Dummy := FALSE;
			Module2101.Output.SkillOutput.SkillOutput0.Error := FALSE;
			Module2101.Output.SkillOutput.SkillOutput0.Ready := FALSE;
			
			//initialize position input with value -1
			IF (NOT GVL.modulePositionInitialized)THEN
				Module2101.Input.PositionInput := -1;
				GVL.modulePositionInitialized := TRUE;
			END_IF
			
			IF (axis.Status.StandStill OR axis.Status.ErrorStop OR axis.Status.Disabled) THEN
				initSubState := step2;	
			END_IF
			
	
	step2:	IF NOT resetAxis.done THEN
				// axreset
				resetAxis (execute := TRUE);
			ELSE
				initSubState := step3;
			END_IF
			
			
	step3:		//Turning Disk clockwise till one of both sensors is detected
				turnDiskSensor(targetVel:= fastVel, sensor:= (iDiskPosition = 2 OR iDiskPosition = 1), execute := TRUE); 
				
				IF (turnDiskSensor.done) THEN
					turnDiskMod(execute:=FALSE);
					initSubState := step4;		
				END_IF
			
	step4:	//turn back to SensorPosition due to lag while stopping
			turnDiskMod(targetPos:= GVL.SensorPosition , targetVel:= fastVel, direction:= Tc2_MC2.MC_Negative_Direction, execute:= TRUE);
			
			IF (turnDiskMod.done AND (iDiskPosition = 2)) THEN
				//if Disk at storage --> step 2	
				initSubState := step5;		
			ELSIF (turnDiskMod.done AND (iDiskPosition = 1)) THEN
				//if Disk at ramp 	 --> step 3
				initSubState := step7;
			END_IF
	
	step5:	//initializing the motor position to a certain value (0)
			setPosition(Axis:= axis, Execute:= FALSE);	//rising edge
			setPosition(Axis:= axis, Execute:= TRUE, Position:= 0, Mode:= FALSE);
			
			initSubState := step6;
			
	step6:	
			//set storage position to 0
			IF (NOT setPosition.Done) THEN
				setPosition(Axis:= axis, Execute:= TRUE, Position:= 0, Mode:= FALSE);
			ELSE
				setPosition(Axis:= axis, Execute:= FALSE);
				GVL.infinitsimu2 := TRUE;
				initSubState := step9;
			END_IF
			
	step7:	//initializing the motor position to a certain value (180)
			setPosition(Axis:= axis, Execute:= FALSE);	//rising edge
			setPosition(Axis:= axis, Execute:= TRUE, Position:= 180, Mode:= FALSE);
			
			initSubState := step8;
			
	step8:		//set storage position to 180
			IF (NOT setPosition.Done) THEN				//set internal Position to 180 (=ramp)
				setPosition(Axis:= axis, Execute:= TRUE, Position:= 180, Mode:= FALSE);
			ELSE
				setPosition(Axis:= axis, Execute:= FALSE);
				infinitsimu := TRUE;		
				initSubState := step9;
			END_IF
			
	
	step9:	//if Cookie is in output --> mainState = ready
			IF (NOT iNoCookieInOutput) THEN					
				GVL.mainState := eMainState.ready;
			ELSE
				//if no Cookie is in output --> mainState = separation
				GVL.mainState := eMainState.separation;	
			END_IF
			initSubState := step0;
END_CASE

END_FUNCTION_BLOCK

// ---- POUs/FB_TurnDiskToSensor.TcPOU
FUNCTION_BLOCK FB_TurnDiskToSensor

VAR_INPUT
	targetVel		: INT;	//Comment here
	sensor			: BOOL;	//Comment here
	execute			: bool;
END_VAR

VAR_OUTPUT
	done 			: BOOL;	//Comment here
END_VAR

VAR
	state		: INT := -10;				//Comment here
	power		: Tc2_MC2.MC_Power;			//Comment here
	turnDisk	: Tc2_MC2.MC_MoveVelocity;	//Comment here
	haltDisk	: Tc2_MC2.MC_Halt;			//Comment here
	
END_VAR

IF (execute) THEN
	power(																		//enable power every cycle
		Axis			:= axis , 
		Enable			:= TRUE , 
		Enable_Positive	:= TRUE , 
		Enable_Negative	:= TRUE , 
		);
	
	CASE state OF 
	 
	-10:	//Comment here
			done := FALSE;

			IF (power.Status AND NOT power.Error) THEN
				state := 0;
			END_IF
		
	0:		//Comment here
			turnDisk(Axis:= axis , Execute:= FALSE);					//rising Edge
			turnDisk(Axis:= axis , Execute:= TRUE, Velocity:=targetVel, Direction:= MC_Positive_Direction);
			state := 10;
			
	10:		//Comment here
			IF (NOT sensor) THEN										//turnDisk until input variable is true
				turnDisk(Axis:= axis);
			
			ELSE 
				GVL.SensorPosition :=axis.NcToPlc.ModuloActPos;				
				turnDisk(Axis:= axis, Execute:= FALSE);
				haltDisk(Axis:= axis, Execute:= TRUE);
				state := 20;
			END_IF
			
	20: 	IF (NOT haltDisk.Done) THEN									//stop turning disk
				haltDisk(Axis:= axis, Execute:= TRUE);
			ELSE
				haltDisk(Axis:= axis, Execute:= FALSE);
				done 	:= TRUE;
				execute := FALSE;
				state	:= -10;
			END_IF
	
	END_CASE

ELSE
	state := -10;
	turnDisk(Axis:= axis , Execute:= FALSE);
END_IF

END_FUNCTION_BLOCK

// ---- POUs/FB_TurnDiskModulo.TcPOU
FUNCTION_BLOCK FB_TurnDiskModulo

VAR_INPUT
	targetPos		: LREAL;
	targetVel		: INT;
	direction		: Tc2_MC2.MC_Direction;
	execute			: BOOL := TRUE;
	
END_VAR

VAR_OUTPUT
	done 			: BOOL;
	turnDisk		: Tc2_MC2.MC_MoveModulo;
END_VAR

VAR
	state		: INT := -10;
	power		: Tc2_MC2.MC_Power;
END_VAR

//Comment here
IF (NOT execute) THEN
	state := -10;
	turnDisk(Axis:= axis , Execute:= FALSE);
ELSE
	//Comment here
	power(
			Axis			:= axis , 
			Enable			:= TRUE , 
			Enable_Positive	:= TRUE , 
			Enable_Negative	:= TRUE , 
			BufferMode		:= Tc2_MC2.MC_BlendingNext
		);				
					
	CASE state OF 
		 
		-10:	//Comment here
				done := FALSE;
				IF (power.Status=TRUE AND power.Error=FALSE) THEN
					state := 0;
				END_IF
							
		0:		//Comment here
				turnDisk(Axis:= axis , Execute:= FALSE);
				turnDisk(Axis:= axis , Execute:= TRUE, Position:= targetPos, Velocity:=targetVel, Direction:= direction, BufferMode:= Tc2_MC2.MC_BlendingNext);
				state := 10;			
				
		10:		//Comment here
				IF (turnDisk.Done=FALSE) THEN
					turnDisk(Axis:= axis, Execute:= TRUE, Position:= targetPos, Velocity:=targetVel, Direction:= direction, BufferMode:= Tc2_MC2.MC_BlendingNext);
				ELSE 
					turnDisk(Axis:= axis, Execute:= FALSE);
					state := 20;
				END_IF
				
		20: 	//Comment here
				done 	:= TRUE;
				execute := FALSE;
				state	:= -10;	
	END_CASE
END_IF

END_FUNCTION_BLOCK

// ---- POUs/FB_Timer.TcPOU
FUNCTION_BLOCK FB_Timer
VAR_INPUT
	iTime	: TIME;
	execute : Bool;
END_VAR
VAR_OUTPUT
	done	: BOOL;
END_VAR
VAR
	timer	: Tc2_Standard.TON;
	state	: INT := 0;
END_VAR

IF (execute) THEN
	
	CASE state OF
	
		0:	done := FALSE;
			timer(IN:= FALSE, PT:= iTime);
			timer(IN:= TRUE, PT:= iTime);
			state := 10;
	
		10:	timer();
			IF (timer.Q) THEN
				done := TRUE;
				state :=0;
			END_IF
	END_CASE

ELSE
	state := 0;
	done := FALSE;
END_IF

END_FUNCTION_BLOCK

// ---- POUs/FB_Output.TcPOU
FUNCTION_BLOCK FB_Output
VAR_INPUT
END_VAR
VAR_OUTPUT
END_VAR
VAR
	turnDiskModFast			: FB_TurnDiskModulo;
	timer					: FB_Timer;
END_VAR

CASE outputSubState OF
	
	step0:	//set OPC state variables
 			Module2101.Output.SkillOutput.SkillOutput0.Ready := FALSE;
			Module2101.Output.SkillOutput.SkillOutput0.Busy := TRUE;
			//reset move functions
			turnDiskModFast(execute := FALSE);
			outputSubState := step1;			

	step1:	//check position of cookie gap
			IF(axis.NcToPlc.ModuloActPos < 5 OR axis.NcToPlc.ModuloActPos > 355) THEN //storage
				outputSubState := step2;
			ELSIF (axis.NcToPlc.ModuloActPos < 182 OR axis.NcToPlc.ModuloActPos > 172) THEN
				outputSubState := step3;
			END_IF
		
	step2:	//turn disk 90° to open clamps and put cookie on XTS mover
			turnDiskModFast(targetPos:= 270, targetVel:= fastVel, direction:= Tc2_MC2.MC_Negative_Direction, execute:= TRUE);
			IF (turnDiskModFast.done) THEN
				outputSubState := step4;
			END_IF
	
	step3:	//turn disk 90° to open clamps and put cookie on XTS mover
			turnDiskModFast(targetPos:= 90, targetVel:= fastVel, direction:= Tc2_MC2.MC_Negative_Direction, execute:= TRUE);
			IF (turnDiskModFast.done) THEN
				outputSubState := step4;
			END_IF
			
	step4:	//tell process tool that cookie is on mover
			Module2101.Output.SkillOutput.SkillOutput0.Busy := FALSE;
			Module2101.Output.SkillOutput.SkillOutput0.Done := TRUE;
			outputSubState := step5;
			
	step5:	// if it was not the first cookie on mover, wait for the XTS to press against iron sheet
			IF (Module2101.Input.SkillInput.SkillInput0.ParameterInput.Parameterinput0.Value = 0) THEN
				outputSubState := step6;
			ELSE
				outputSubState := step7;
			END_IF
			timer(execute := FALSE);
			
	step6:	//waiting time if not first cookie
			timer(iTime:= T#5S, execute:= TRUE);
			IF (timer.done) THEN
				outputSubState := step7;
				timer(execute := FALSE);
			END_IF
			
	step7:	//OPC UA communication
			IF (NOT Module2101.Input.SkillInput.SkillInput0.Execute) THEN
				Module2101.Output.SkillOutput.SkillOutput0.Done := FALSE;
				outputSubState := step8;
			END_IF
			
	step8:	//change into separation state
			mainState := eMainState.separation;	
			outputSubState := step0;
END_CASE

END_FUNCTION_BLOCK

// ---- POUs/FB_Ready.TcPOU
FUNCTION_BLOCK FB_Ready
VAR_INPUT
END_VAR
VAR_OUTPUT
END_VAR
VAR
	execute : bool := false;
END_VAR

IF (NOT (Module2101.Input.PositionInput = -1)) THEN
	
	//set OPC UA variable -> state ready
	Module2101.Output.SkillOutput.SkillOutput0.Ready := TRUE;
	
	//wait for execute signal and the n change state to output
	IF(Module2101.Input.SkillInput.SkillInput0.Execute) THEN
		//order received
		Module2101.Output.SkillOutput.SkillOutput0.Ready := FALSE;
		mainState:=eMainState.output;
	END_IF

END_IF

END_FUNCTION_BLOCK

// ---- POUs/FB_Refill.TcPOU
FUNCTION_BLOCK FB_Refill
VAR_INPUT
END_VAR
VAR_OUTPUT
END_VAR
VAR
END_VAR

CASE refillSubState OF

	step0:	//go in the right error state
			Module2101.Output.CurrentTaskDescription := 'CookieStorage empty. Switching to refill mode.';
			Module2101.Output.ErrorID := 1;
			Module2101.Output.Error := TRUE;
			Module2101.Output.ErrorDescription := 'storage empty. please refill';
			
			//wait for process tool to set the module in manual mode
			IF(Module2101.Input.Mode = DUT_MODE.Manual) THEN
				refillSubState := step1;
			END_IF
			
	step1:	//wait for process tool to set the module in init mode
			IF(Module2101.Input.Mode = DUT_MODE.Auto) THEN
				//reset error 
				Module2101.Output.Error := FALSE;
				Module2101.Output.ErrorDescription := '';
				Module2101.Output.ErrorID := 0;
				
				//change to init state
				initSubState := step0;
				mainState := eMainState.init;
				refillSubState := step0;
			END_IF
END_CASE

END_FUNCTION_BLOCK

// ---- POUs/FB_ResetSystem.TcPOU
FUNCTION_BLOCK FB_ResetSystem
VAR_INPUT
END_VAR
VAR_OUTPUT
END_VAR
VAR
	resetAxis : FB_ResetAxis;
END_VAR

CASE GVL.resetSubState OF

step0:	resetAxis (execute := FALSE);

		Module2101.Output.SkillOutput.SkillOutput0.Busy := TRUE;
		Module2101.Output.SkillOutput.SkillOutput0.Done := TRUE;
		Module2101.Output.SkillOutput.SkillOutput0.Error := TRUE;
		Module2101.Output.SkillOutput.SkillOutput0.Ready := TRUE;
		
		GVL.resetSubState := step1;
		
step1:	IF NOT resetAxis.done THEN
		// axreset
		resetAxis (execute := TRUE);
		ELSE
			GVL.resetSubState := step2;
		END_IF
		
step2:	// reset substates
		GVL.refillSubState := step0;
		GVL.separationSubState := step0;
		GVL.outputSubState := step0;
		GVL.emergencySubState := step0;
		GVL.errorSubState := step0;
		GVL.initSubState := step0;
		
		GVL.resetSubState := step0;
		
		MI5.reset := FALSE;
		GVL.mainState := eMainState.init;	
		
END_CASE

END_FUNCTION_BLOCK

// ---- POUs/FB_Separation.TcPOU
FUNCTION_BLOCK FB_Separation
VAR_INPUT
END_VAR
VAR_OUTPUT
END_VAR
VAR
	turnDiskModFast			: FB_TurnDiskModulo;
	turnDiskModSlow			: FB_TurnDiskModulo;
	storageLevel			: FB_StorageLevel;
	timer					: FB_Timer;
	timer2					: FB_Timer;
	
	counter					: INT := 1;
	cookieBroken			: INT := 100;
	
END_VAR

CASE separationSubState OF

	step0:	//set OPC state variables
			Module2101.Output.SkillOutput.SkillOutput0.Busy := TRUE;
			//reset all move functions
			turnDiskModFast(execute := FALSE);
			turnDiskModSlow(execute := FALSE);
			
			//check if possible to separate
			IF (GVL.empty) THEN
				//you have to refill
				mainState:=eMainState.refill;	
			ELSE
			separationSubState:=step1;
			END_IF

	step1:	//check/bring cookieGap to storage
			IF (axis.NcToPlc.ModuloActPos < 5 OR axis.NcToPlc.ModuloActPos > 355) THEN
				separationSubState := step3;
			ELSE
				//move cookieGap to storage
				separationSubState := step2;
			END_IF
			
	step2:	//move cookieGap to storage in anti-clockwise to ensure the gap is empty
			turnDiskModFast(targetPos:= 0, targetVel:= fastVel, direction:= Tc2_MC2.MC_Negative_Direction, execute:= TRUE);
			IF (turnDiskModFast.done) THEN
				separationSubState := step3;
			END_IF
			
	step3:	//move cookieGap to wenglor camera test (280°) 
			IF (MI5.cameraFix) THEN
				separationSubState := step8;
			ELSE
				turnDiskModFast(targetPos:= 276, targetVel:= fastVel, direction:= Tc2_MC2.MC_Negative_Direction, execute:= TRUE);
				IF (turnDiskModFast.done) THEN
					separationSubState := step4;
					timer(execute:= FALSE);
				END_IF
			END_IF
			
	step4:	// check if cookie is broken or not (getting from cameraDetection)
			timer(iTime:= T#1S, execute:= TRUE);
			IF(timer.done) THEN
				separationSubState := step5;
				timer(execute:= FALSE);
			END_IF;
			
	step5:	GVL.oTriggerCamera := TRUE;
			timer2(iTime:= T#60MS, execute:= TRUE);
			IF (timer2.done) THEN
				GVL.oTriggerCamera := FALSE;
				separationSubState := step6;
				timer2(execute:= FALSE);
			END_IF
			
	step6:	IF (counter < 10) THEN
				counter := counter + 1;
				IF (NOT iCookieIntact) THEN
					cookieBroken := cookieBroken - 1;	
				ELSIF (iCookieIntact) THEN
						cookieBroken := cookieBroken + 1;		
				END_IF
				separationSubState := step5;
			ELSE	
				IF (cookieBroken < 100) THEN
					separationSubState := step7;	
				ELSIF (cookieBroken >= 100) THEN
					separationSubState := step8;		
				END_IF
			END_IF
			
	step7:	// move cookieGap to the broken cookie output hole (backwards)
			cookieBroken := 100;
			counter := 1;
			turnDiskModFast(targetPos:= 90, targetVel:= fastVel, direction:= Tc2_MC2.MC_Positive_Direction, execute:= TRUE);
			IF(turnDiskModFast.done) THEN
				separationSubState := step0;
				// start with separation from beginning
			END_IF
			
	step8:	// move cookieGap to the start of the mechanical broken cookie output (fast velocity)
			cookieBroken := 100;
			counter := 1;
			turnDiskModFast(targetPos:= 200, targetVel:= fastVel, direction:= Tc2_MC2.MC_Negative_Direction, execute:= TRUE);
			IF(turnDiskModFast.turnDisk.Active) THEN
				separationSubState := step9;
			END_IF	
			
	step9:	// move cookieGap to the end of the mechanical broken cookie output (slow velocity)
			turnDiskModSlow(targetPos:= 178, targetVel:= slowVel, direction:= Tc2_MC2.MC_Negative_Direction, execute:= TRUE);
			IF(turnDiskModSlow.turnDisk.Done) THEN
				turnDiskModFast(execute:=FALSE);
				turnDiskModSlow(execute:=FALSE);
				separationSubState := step10;
			END_IF
			
	step10:	// move cookieGap to the ramp(fast)
			turnDiskModSlow(targetPos:= 180, targetVel:= slowVel, direction:= Tc2_MC2.MC_Positive_Direction, execute:= TRUE);
			IF(turnDiskModSlow.done) THEN
				separationSubState := step11;
			END_IF
			
	step11:	// wait 5s for cookie to slide down the ramp
			//@TODO: test how long cookie needs to slide down
			//@TODO: implement error case if the cookie gets stuck on ramp
			turnDiskModSlow(execute:=FALSE);
			timer(iTime:=T#3S, execute := TRUE);
			IF(timer.done) THEN
				separationSubState := step12;
				timer2(execute:= FALSE);
			END_IF
			
	step12:	//check if cookie is in output, if not start from beginning
			IF(NOT iNoCookieInOutput) THEN
				Module2101.Output.SkillOutput.SkillOutput0.Busy := FALSE;
				mainState := eMainState.ready;
			END_IF
			separationSubState := step0;
END_CASE

END_FUNCTION_BLOCK

// ---- POUs/FB_StorageLevel.TcPOU
FUNCTION_BLOCK FB_StorageLevel
VAR_INPUT
END_VAR
VAR_OUTPUT
END_VAR
VAR
	calculatedCookies		: LREAL;
	remainingCookies 		: INT;	
END_VAR

//Comment here	
IF (GVL.iStorageLevel > 226000) THEN
    GVL.empty:=TRUE;
	remainingCookies := 0;
// configuration for all cookies (not as acurate)
ELSE
    GVL.empty:=FALSE;
	calculatedCookies := (231000 - GVL.iStorageLevel)/5247;
	remainingCookies := REAL_TO_INT(calculatedCookies);
END_IF


Module2101.Output.StateValue.StateValue0.Name := 'Remaining cookies';
Module2101.Output.StateValue.StateValue0.Description := 'Number of remaining cookies in storage.';
Module2101.Output.StateValue.StateValue0.Dummy := FALSE;
Module2101.Output.StateValue.StateValue0.Value := remainingCookies;

IF (remainingCookies = 1) THEN
	Module2101.Output.StateValue.StateValue0.Unit := 'Cookie';
ELSE
	Module2101.Output.StateValue.StateValue0.Unit := 'Cookies';
END_IF

(*

//configuration for bright cookies
ELSE
    empty:=FALSE;
	calculatedCookies := (231000 - GVL.iStorageLevel)/5129;
	remainingCookies := REAL_TO_INT(calculatedCookies);
END_IF;

//configuration for dark cookies
ELSE
    empty:=FALSE;
	calculatedCookies := (231000 - GVL.iStorageLevel)/5366;
	remainingCookies := REAL_TO_INT(calculatedCookies);
END_IF;

*)

END_FUNCTION_BLOCK

// ---- POUs/MAIN.TcPOU
PROGRAM MAIN
VAR											//FBI = function block instance
	FBI_init			: FB_Init;			//Comment here	
	FBI_output			: FB_Output;		//Comment here	
	FBI_refill			: FB_Refill;		//Comment here	
	FBI_separation		: FB_Separation;	//Comment here	
	FBI_ready			: FB_Ready;			//Comment here	
	FBI_emergencyStop 	: FB_EmergencyStop;	//Comment here	
	FBI_error 			: FB_error;			//Comment here	
	FBI_storageLevel	: FB_StorageLevel;	//Comment here
	FBI_resetSystem		: FB_ResetSystem;  
	
	//Interface variables:
	FBI_Timer			: TOF;				//Comment here	
		
END_VAR

// @TODO measure position of slide against position sensor of XTS

//----------------------------------------- Error handling and emergency stop ------------------------------------------
axis.ReadStatus();

//reset system
IF (Mi5.reset) THEN
	GVL.mainState := eMainState.resetSystem;
	
//Emergency Stop Watchdog!
ELSIF Module2101.Input.EmergencyStop THEN
	GVL.mainState := eMainState.emergencyStop;

//error handling
ELSIF (axis.Status.Error) THEN
	GVL.mainState := eMainState.error;

END_IF

//------------------------------------------------ OPC UA and module init --------------------------------------------------------------

//Connection Test
Module2101.Output.ConnectionTestOutput := Module2101.Input.ConnectionTestInput;
//positionsweitergabe an process tool
Module2101.Output.PositionOutput := Module2101.Input.PositionInput + 143; 

//module positioning (by fj)
FBI_Timer();
IF GVL.init_sensor THEN
	Module2101.Output.PositionSensor := TRUE;
	FBI_Timer(IN := TRUE,PT := T#400MS);
	FBI_Timer(IN := FALSE,PT := T#400MS);
ELSE
	Module2101.Output.PositionSensor := FBI_Timer.Q;
END_IF

//----------------------------------------------- cookie function process and parameter reading ----------------------------------------------------

//calculate storage level
FBI_storageLevel();


//----------------------------------------------- pseudo function block calls ----------------------------------------------------------------------
CASE GVL.mainState OF

	eMainState.init: //<<<<<<<<<<<<<<<<<<<<<<<<<<<<<<<<<<<<<<<<<<<<<<<<<<<<<<<<<<<<<<
		//init of state whereever the position of the disk is
		FBI_init();				
	
	eMainState.ready: //<<<<<<<<<<<<<<<<<<<<<<<<<<<<<<<<<<<<<<<<<<<<<<<<<<<<<<<<<<<<<
		//cookie is on the clamps, waiting for putting it on the mover
		FBI_ready();
		
	eMainState.output: //<<<<<<<<<<<<<<<<<<<<<<<<<<<<<<<<<<<<<<<<<<<<<<<<<<<<<<<<<<<<<
		//now open the clamps and let the cookie go down
		FBI_output();

	eMainState.refill: //<<<<<<<<<<<<<<<<<<<<<<<<<<<<<<<<<<<<<<<<<<<<<<<<<<<<<<<<<<<<
		//cookie storage empty --> needs to be refilled
		FBI_refill();
	
	eMainState.separation:	//<<<<<<<<<<<<<<<<<<<<<<<<<<<<<<<<<<<<<<<<<<<<<<<<<<<<<<<
		//take a new cookie and bring it to the output clamps
		FBI_separation();
		
	eMainState.emergencyStop: //<<<<<<<<<<<<<<<<<<<<<<<<<<<<<<<<<<<<<<<<<<<<<<<<<<<<<<<<<<<<
		// manually set emergency stop
		FBI_emergencyStop();
		
	eMainState.error: //<<<<<<<<<<<<<<<<<<<<<<<<<<<<<<<<<<<<<<<<<<<<<<<<<<<<<<<<<<<<
		//error state
		FBI_error(); 
		
	eMainState.resetSystem: //<<<<<<<<<<<<<<<<<<<<<<<<<<<<<<<<<<<<<<<<<<<<<<<<<<<<<<<<<<<<
		//error state
		FBI_resetSystem(); 

END_CASE

END_PROGRAM
